FUNCTION_BLOCK "Siemens_vav_compact_controller"   // FB60, SCL
{ S7_Optimized_Access := 'TRUE' }
VERSION : 0.1
   VAR_INPUT
      mb_addr : UInt;
      sp : Real;   // setpoint
      sp_backup : Real;
   END_VAR
   VAR_IN_OUT
      mb_query : "mb_query";
   END_VAR
   VAR
      sb : "mb_station_block_udt";
      read : Struct
         Actual_position : Int;
         Actual_Flow_rel : UInt;
         Actual_Flow_abs : UInt;
         Actual_Pressure : UInt;
      END_STRUCT;
      write1 : Struct
         Setpoint : Int;
      END_STRUCT;
      write2 : Struct
         backup_mode : Int;
         backup_position : Int;
      END_STRUCT;
   END_VAR
BEGIN
   // Siemens - VAV compact controller 
   // GDB181.1E/MO Operating voltage AC 24 V, 5 Nm
   // GLB181.1E/MO Operating voltage AC 24 V, 10 Nm

   // https://www.micromatic.no/globalassets/inriver/resources/
   // bruksanvisning_ko1320-28.pdf

   "mb_station_block_header"(sb := #sb, mb_query := #mb_query);
   #mb_query.mb_addr := #mb_addr;

   #mb_query.mode := #mb_query.c.read.holding_reg;
   #mb_query(data_addr := 3, data_ptr := #read);

   #mb_query.mode := #mb_query.c.write.holding_reg;
   #write1.Setpoint := REAL_TO_INT(#sp) * 100;
   #mb_query(data_addr := 1, data_ptr := #write1);
   #write2.backup_position := REAL_TO_INT(#sp_backup) * 100;
   #mb_query(data_addr := 513, data_ptr := #write2);

   "mb_station_block_footer"(sb := #sb, mb_query := #mb_query);

   (*
   Backup mode (write 2)
   0 = Go to BackupPosition
   1 = Keep last position
   2 = Disabled
   *)
END_FUNCTION_BLOCK

FUNCTION_BLOCK "Siemens_SIWAREX_WP251"   // FB93, SCL
{ S7_Optimized_Access := 'TRUE' }
VERSION : 0.1
   VAR_INPUT
      mb_addr : UInt;
   END_VAR
   VAR_IN_OUT
      mb_query : "mb_query";
   END_VAR
   VAR
      sb : "mb_station_block_udt";
      read1 : Struct
         Unit_of_weight : UInt;   // x1000
         Gross_identifier : UInt;
         Code_for_regulations : UInt;
         Reserve : UInt;
         weighing_range_min : UInt;
         weighing_range_max : Real;
         Calibration_weight : Array[0..2] of Real;
         Calibration_digits : Array[0..2] of Real;
         Scale_interval : Array[0..2] of Real;   // (Page 64)
      END_STRUCT;
      read2 : Struct
         stat : Struct
            x08 : Bool;
            x09 : Bool;
            x10 : Bool;
            x11 : Bool;
            x12 : Bool;
            x13 : Bool;
            x14 : Bool;
            x15 : Bool;
            x00 : Bool;
            x01 : Bool;
            x02 : Bool;
            x03 : Bool;
            x04 : Bool;
            x05 : Bool;
            x06 : Bool;
            x07 : Bool;
         END_STRUCT;
         Reserve : UInt;
         Max_tare_load : Real;
         Max_negative_zero_limit_power_on : Real;
         Max_positive_zero_limit_power_on : Real;
         Max_negative_zero_limit_semi_automatically : Real;
         Max_positive_zero_limit_semi_automatically : Real;
      END_STRUCT;
      read3 : Struct
         standstill : Array[1..2] of Struct
            range : Real;
            "time" : Time;
            max_waiting_time : Time;
         END_STRUCT;
         frequency_low_pass_filter1 : Real;
         Order_no_low_pass_filter1 : UInt;
         depth_average_filter : UInt;
         reserve_1 : UInt;
         weighing_operating_mode : UInt;
         resolution_of_master_totalizer : Real;
         Reserve_2 : Real;
         SecureDisplay_including_weighing_range_data : UInt;
      END_STRUCT;
      read4 : Struct
         SecureDisplay_interface : UInt;   // (Page 71)
         String_header_version_SecureDisplay : String[2];
         SecureDisplay_version : String[12];
         Minimum_zoom_factor_of_SecureDisplay : UInt;
         Reserve_1 : Array[1..3] of Real;
         Reserve_2 : Array[1..3] of UInt;
         Grid_frequency : UInt;   // 0: 50 Hz, 1: 60Hz
      END_STRUCT;
      write1 : Struct
         Smallest_weight_below_TU2 : Real;
         Highest_weight_above_TH2 : Real;
         Single_setpoin : Real;
         Net_weight_average_value : Real;
         Standard_deviation : Real;
      END_STRUCT;
   END_VAR
BEGIN
   // Siemens - SIWAREX WP251 - Electronic Weighing System
   // A5E37203357A
   // 
   // https://cache.industry.siemens.com/dl/files/751/109481751/att_893477/v1/Manual_SIWAREX_WP251_en_en-US.pdf

   "mb_station_block_header"(sb := #sb, mb_query := #mb_query);
   #mb_query.mb_addr := #mb_addr;

   #mb_query.mode := #mb_query.c.read.holding_reg;
   #mb_query(data_addr := 1011, data_ptr := #read1);
   #mb_query(data_addr := 1032, data_ptr := #read2);
   #mb_query(data_addr := 1044, data_ptr := #read3);
   #mb_query(data_addr := 1067, data_ptr := #read4);

   #mb_query.mode := #mb_query.c.write.holding_reg;
   #mb_query(data_addr := 4101, data_ptr := #write1);

   "mb_station_block_footer"(sb := #sb, mb_query := #mb_query);

   (*
   Unit of weight:
   0: "mg"
   1: "g"
   2: "kg"
   3: "t"
   4: "oz" (ounce)
   5: "lb" (pound)
   6: "T" (=short tons)
   7: "TL" (= long tons)

   Gross identifier:
   0: "brutto" 
   1: "Gross"

   Code for regulations:
   0: None
   1: OIML

   Weighing operating mode (Page 71):
   0: NAWI – Filling
   1: NAWI – Removal
   10: AWI
   20: ACI – Filling 
   21: ACI – Removal

   *)
END_FUNCTION_BLOCK

// folder: Library/Modbus/Station blocks/sb untested/Swan

FUNCTION_BLOCK "Swan_AMI_CACE"   // FB65, SCL
{ S7_Optimized_Access := 'TRUE' }
VERSION : 0.1
   VAR_INPUT
      mb_addr : USInt;
   END_VAR
   VAR_IN_OUT
      mb_query : "mb_query";
   END_VAR
   VAR
      sb : "mb_station_block_udt";
      data : Struct
         cond_sc : Array[1..3] of Real;   // µS
         Temp : Array[1..3] of Real;
         flow : Real;
         pH : Real;
         alkalyzer : Real;
         cond_uc : Array[1..3] of Real;
         Pt1000_Temp : Array[1..3] of Real;
         raw_flow : Real;
         case_temperature : Real;
         EDI_voltage : Real;
         EDI_current : Real;
         Degasser_temperature : Real;
         Degasser_boiling_point : Real;
         Degasser_PWM : Real;
         Degasser_line_voltage : Real;
         Degasser_air_pressure : Real;
         Degasser_Case_Temp : Real;
         signal_output : Array[1..2] of Real;
         "Instrument Display Status" : DWord;
      END_STRUCT;
      alarm : Struct
         x00_Cond_1_Alarm_high : Bool;
         x01_Cond_1_Alarm_low : Bool;
         x02_Cond_2_Alarm_high : Bool;
         x03_Cond_2_Alarm_low : Bool;
         x04_Cond_3_Alarm_high : Bool;
         x05_Cond_3_Alarm_low : Bool;
         x06_Temp_1_high : Bool;
         x07_Temp_1_low : Bool;
         x08_sample_flow_high : Bool;
         x09_sample_flow_low : Bool;
         x10_temp_1_shorted : Bool;
         x11_temp_1_disconnected : Bool;
         x12_case_temp_high : Bool;
         x13_case_temp_low : Bool;
         x14_pH_Error : Bool;
         x15_Degasser_frontend : Bool;
         x16_control_timeout : Bool;
         x17_Degasser_disconnected : Bool;
         x18_Temp_2_shorted : Bool;
         x19_Temp_2_disconnected : Bool;
         x20_Temp_3_shorted : Bool;
         x21_Temp_3_disconnected : Bool;
         x22_Degasser_Ctl_Timeout : Bool;
         x23_Input_Active : Bool;
         x24_IC_MK41T56 : Bool;
         x25_IC_LM75 : Bool;
         x26_IC_PCF8574 : Bool;
         x27_Signal_output_open : Bool;
         x28_Calibration_Degasser : Bool;
         x29_EEprom_Front_end : Bool;
         x30_Calibration_Recout : Bool;
         x31_Wrong_Front_end : Bool;
         x32_pH_Alarm_high : Bool;
         x33_pH_Alarm_low : Bool;
         x34_Alkali_Alarm_high : Bool;
         x35_Alkali_Alarm_low : Bool;
         x36_Temp_2_high : Bool;
         x37_Temp_2_low : Bool;
         x38_Temp_3_high : Bool;
         x39_Temp_3_low : Bool;
         x40_Degasser_Line_Voltage : Bool;
         x41_Degasser_Temperature : Bool;
         x42_EDI_out_of_range : Bool;
         x43_No_sample_flow : Bool;
         x44_EDI_DAC_disconnected : Bool;
         "x45_ EDI_ADC_disconnected" : Bool;
         x46 : Bool;
         x47_EDI_module_exhausted : Bool;
      END_STRUCT;
      write : Struct
         x0_relay_contacts_1 : Bool;
         x1_relay_contacts_2 : Bool;
         x2 : Bool;
         x3 : Bool;
         x4 : Bool;
         x5 : Bool;
         x6 : Bool;
         x7 : Bool;
      END_STRUCT;
   END_VAR
BEGIN
   // Swan - AMI CACE - Conductivity measurement 
   // Swan analytical instruments
   // http://www.swan.ch/GetAttachment.axd?attaName=e82f8e94-ab32-4930-8c9d-a56dc0847f61
   // Page 9

   "mb_station_block_header"(sb := #sb,
                             mb_query := #mb_query);
   #mb_query.mb_addr := #mb_addr;
   #mb_query.data_addr := 0;

   #mb_query(mode := #mb_query.c.read.input_reg,
             data_ptr := #data);

   #mb_query(mode := #mb_query.c.read.discrete_input,
             data_ptr := #alarm);

   (*#mb_query(mode := #mb_query.c.write.discrete_output,
             data_len := 2,
             data_ptr := #write);*)

   "mb_station_block_footer"(sb := #sb,
                             mb_query := #mb_query);
END_FUNCTION_BLOCK

FUNCTION_BLOCK "Swan_AMI_Codes-II_CC"   // FB66, SCL
{ S7_Optimized_Access := 'TRUE' }
VERSION : 0.1
   VAR_INPUT
      mb_addr : USInt;
   END_VAR
   VAR_IN_OUT
      mb_query : "mb_query";
   END_VAR
   VAR
      sb : "mb_station_block_udt";
      data : Struct
         free_available_chlorine : Real;   // ppm
         total_chlorine_1_tc1 : Real;   // ppm
         total_chlorine_2_tc2 : Real;   // ppm
         calculated_monochloramine : Real;   // ppm
         calculated_combined_chlorine : Real;   // ppm
         calculated_dichloramine : Real;   // ppm
         temperature : Real;   // °C
         flow : Real;   // B/s
         pH : Real;   // pH
         absorbance : Real;
         photometer_frequency : Real;   // Hz
         remaining_DPD_buffer : Real;   // %
         remaining_potassium_Iodide : Real;   // %
         remaining_cleaning_solution : Real;   // %
         raw_temp_NTK5 : Real;   // Ohm
         raw_flow : Real;   // Hz
         raw_pH : Real;   // mV
         case_temperature : Real;   // °C
         signal_output_1 : Real;   // mA
         signal_output_2 : Real;   // mA
         instrument_display_status : Real;
      END_STRUCT;
      alarm : Struct
         x00_high_fac : Bool;
         x01_low_fac : Bool;
         x02_high_tc1 : Bool;
         x03_low_tc1 : Bool;
         x04_high_tc2 : Bool;
         x05_low_tc2 : Bool;
         x06_sample_temp_high : Bool;
         x07_sample_temp_low : Bool;
         x08_sample_flow_high : Bool;
         x09_sample_flow_low : Bool;
         x10_Temp_shorted : Bool;
         x11_Temp_disconnected : Bool;
         x12_case_temp_high : Bool;
         x13_case_temp_low : Bool;
         x14_valve_1_defective : Bool;
         x15_dis_invalid : Bool;
         x16_control_timeout : Bool;
         x17_reagent_pump : Bool;
         x18_photometer_not_connected : Bool;
         x19_photometer_dirty : Bool;
         x20_absorbance_too_high : Bool;
         x21_reagent_empty : Bool;
         x22_cleaning_reagent : Bool;
         x23_input_active : Bool;
         x24_IC_MK41T56 : Bool;
         x25_IC_LM75 : Bool;
         x26_IC_PCF8574 : Bool;
         x27_signal_output_open : Bool;
         x28_EEprom_motherboard : Bool;
         x29_EEprom_front_end : Bool;
         x30_calibration_recout : Bool;
         x31_wrong_front_end : Bool;
         x32_high_cmc : Bool;
         x33_low_cmc : Bool;
         x34_high_ccc : Bool;
         x35_low_ccc : Bool;
         x36_high_cdc : Bool;
         x37_low_cdc : Bool;
         x38_high_pH : Bool;
         x39_low_pH : Bool;
         x40_DPD_buffer : Bool;
         x41_potassium_Iodide : Bool;
         x42_cleaning_solution : Bool;
         x43 : Bool;
         x44 : Bool;
         x45 : Bool;
         x46 : Bool;
         x47 : Bool;
      END_STRUCT;
      write : Struct
         x0_relay_contacts_1 : Bool;
         x1_relay_contacts_2 : Bool;
         x2_hold : Bool;
         x3_Remote_off : Bool;
         x4 : Bool;
         x5 : Bool;
         x6 : Bool;
         x7 : Bool;
      END_STRUCT;
   END_VAR
BEGIN
   // Swan - AMI Codes-II CC
   //
   // http://www.swan.ch/GetAttachment.axd?attaName=e82f8e94-ab32-4930-8c9d-a56dc0847f61
   // Page 17

   "mb_station_block_header"(sb := #sb,
                             mb_query := #mb_query);
   #mb_query.mb_addr := #mb_addr;
   #mb_query.data_addr := 0;

   #mb_query(mode := #mb_query.c.read.input_reg,
             data_ptr := #data);

   #mb_query(mode := #mb_query.c.read.discrete_input,
             data_ptr := #alarm);

   (*#mb_query(mode := #mb_query.c.write.discrete_output,
             data_len := 4,
             data_ptr := #write);*)

   "mb_station_block_footer"(sb := #sb,
                             mb_query := #mb_query);
END_FUNCTION_BLOCK

FUNCTION_BLOCK "Swan_AMI_Hydrogen"   // FB67, SCL
{ S7_Optimized_Access := 'TRUE' }
VERSION : 0.1
   VAR_INPUT
      mb_addr : USInt;
   END_VAR
   VAR_IN_OUT
      mb_query : "mb_query";
   END_VAR
   VAR
      sb : "mb_station_block_udt";
      data : Struct
         hydrogen : Real;   // ppb
         temperature : Real;   // °C
         flow : Real;   // l/h
         saturation : Real;   // %
         air_pressure : Real;   // hPa
         raw_Current_temp_compensated : Real;   // nA
         raw_current_uncompensated : Real;   // nA
         raw_temp_Pt1000 : Real;   // Ω
         raw_flow : Real;   // Hz
         reserved : Real;
         case_temperature : Real;   // °C
         signal_output_1 : Real;   // mA
         signal_output_2 : Real;   // mA
         instrument_display_status : UDInt;
      END_STRUCT;
      alarm : Struct
         x00_hydrogen_alarm_high : Bool;
         x01_hydrogen_alarm_low : Bool;
         x02_saturation_alarm_high : Bool;
         x03_saturation_alarm_low : Bool;
         x04 : Bool;
         x05 : Bool;
         x06_sample_temp_high : Bool;
         x07_sample_temp_low : Bool;
         x08_sample_flow_high : Bool;
         x09_sample_flow_low : Bool;
         x10_temp_shorted : Bool;
         x11_temp_disconnected : Bool;
         x12_case_temp_high : Bool;
         x13_case_temp_low : Bool;
         x14 : Bool;
         x15 : Bool;
         x16_control_timeout : Bool;
         x17_faraday_efficiency_QED : Bool;
         x18_quality_assurance : Bool;
         x19 : Bool;
         x20 : Bool;
         x21 : Bool;
         x22 : Bool;
         x23_input_active : Bool;
         x24_IC_MK41T56 : Bool;
         x25_IC_LM75 : Bool;
         x26_IC_PCF8574 : Bool;
         x27_Signal_output_open : Bool;
         x28_EEprom_Motherboard : Bool;
         x29_EEprom_Front_end : Bool;
         x30_Calibration_Recout : Bool;
         x31_Wrong_Front_end : Bool;
         x32 : Bool;
         x33 : Bool;
         x34 : Bool;
         x35 : Bool;
         x36 : Bool;
         x37 : Bool;
         x38 : Bool;
         x39 : Bool;
         x40 : Bool;
         x41 : Bool;
         x42 : Bool;
         x43 : Bool;
         x44 : Bool;
         x45 : Bool;
         x46 : Bool;
         x47_Status_Electrolyte_depleted : Bool;
      END_STRUCT;
      write : Struct
         x0_relay_contacts_1 : Bool;
         x1_relay_contacts_2 : Bool;
         x2_hold : Bool;
         x3_Remote_off : Bool;
         x4 : Bool;
         x5 : Bool;
         x6 : Bool;
         x7 : Bool;
      END_STRUCT;
   END_VAR
BEGIN
   // Swan - AMI Hydrogen
   // Swan analytical instruments
   // http://www.swan.ch/GetAttachment.axd?attaName=e82f8e94-ab32-4930-8c9d-a56dc0847f61
   // Page 37

   "mb_station_block_header"(sb := #sb,
                             mb_query := #mb_query);
   #mb_query.mb_addr := #mb_addr;
   #mb_query.data_addr := 0;

   #mb_query(mode := #mb_query.c.read.input_reg,
             data_ptr := #data);

   #mb_query(mode := #mb_query.c.read.discrete_input,
             data_ptr := #alarm);

   (*#mb_query(mode := #mb_query.c.write.discrete_output,
             data_len := 4,
             data_ptr := #write);*)

   "mb_station_block_footer"(sb := #sb,
                             mb_query := #mb_query);
END_FUNCTION_BLOCK

FUNCTION_BLOCK "Swan_AMI_Oxysafe"   // FB68, SCL
{ S7_Optimized_Access := 'TRUE' }
VERSION : 0.1
   VAR_INPUT
      mb_addr : USInt;
   END_VAR
   VAR_IN_OUT
      mb_query : "mb_query";
   END_VAR
   VAR
      sb : "mb_station_block_udt";
      data : Struct
         oxygen : Real;   // ppm
         temperature : Real;   // °C
         flow : Real;   // l/h
         saturation : Real;   // %
         air_pressure : Real;   // hPa
         raw_Oxygen_temp_compensated : Real;   // nA
         raw_oxygen_temp_uncompensated : Real;   // nA
         raw_Temp_Pt1000 : Real;   // Ohm
         raw_flow : Real;   // Hz
         remaining_electrolyte : Real;   // %
         case_temperature : Real;   // °C
         signal_output_1 : Real;   // mA
         signal_output_2 : Real;   // mA
         instrument_display_status : DWord;
      END_STRUCT;
      alarm : Struct
         x00_Oxygen_alarm_high : Bool;
         x01_Oxygen_alarm_low : Bool;
         x02_Saturation_alarm_high : Bool;
         x03_Saturation_alarm_low : Bool;
         x04 : Bool;
         x05 : Bool;
         x06_Sample_temp_high : Bool;
         x07_Sample_temp_low : Bool;
         x08_sample_flow_high : Bool;
         x09_sample_flow_low : Bool;
         x10_temp_shorted : Bool;
         x11_temp_disconnected : Bool;
         x12_case_temp_high : Bool;
         x13_case_temp_low : Bool;
         x14 : Bool;
         x15 : Bool;
         x16_control_timeout : Bool;
         x17_Faraday_efficiency_QED : Bool;
         x18 : Bool;
         x19 : Bool;
         x20 : Bool;
         x21 : Bool;
         x22 : Bool;
         x23_input_active : Bool;
         x24_IC_MK41T56 : Bool;
         x25_IC_LM75 : Bool;
         x26_IC_PCF8574 : Bool;
         x27_Signal_output_open : Bool;
         x28_EEprom_Motherboard : Bool;
         x29_EEprom_Front_end : Bool;
         x30_Calibration_Recout : Bool;
         x31_Wrong_Front_end : Bool;
         x32 : Bool;
         x33 : Bool;
         x34 : Bool;
         x35 : Bool;
         x36 : Bool;
         x37 : Bool;
         x38 : Bool;
         x39 : Bool;
         x40_Electrolyte_depleted : Bool;
         x41 : Bool;
         x42 : Bool;
         x43 : Bool;
         x44 : Bool;
         x45 : Bool;
         x46 : Bool;
         x47 : Bool;
      END_STRUCT;
      write : Struct
         x0_relay_contacts_1 : Bool;
         x1_relay_contacts_2 : Bool;
         x2_hold : Bool;
         x3_Remote_off : Bool;
         x4 : Bool;
         x5 : Bool;
         x6 : Bool;
         x7 : Bool;
      END_STRUCT;
   END_VAR
BEGIN
   // Swan - AMI - Oxysafe
   // Swan analytical instruments
   // http://www.swan.ch/GetAttachment.axd?attaName=e82f8e94-ab32-4930-8c9d-a56dc0847f61
   // Page 53

   "mb_station_block_header"(sb := #sb,
                             mb_query := #mb_query);
   #mb_query.mb_addr := #mb_addr;
   #mb_query.data_addr := 0;

   #mb_query(mode := #mb_query.c.read.input_reg,
             data_ptr := #data);

   #mb_query(mode := #mb_query.c.read.discrete_input,
             data_ptr := #alarm);

   (*#mb_query(mode := #mb_query.c.write.discrete_output,
             data_len := 4,
             data_ptr := #write);*) 

   "mb_station_block_footer"(sb := #sb,
                             mb_query := #mb_query);
END_FUNCTION_BLOCK

FUNCTION_BLOCK "Swan_AMI_pH-Redox"   // FB69, SCL
{ S7_Optimized_Access := 'TRUE' }
VERSION : 0.1
   VAR_INPUT
      mb_addr : USInt;
   END_VAR
   VAR_IN_OUT
      mb_query : "mb_query";
   END_VAR
   VAR
      sb : "mb_station_block_udt";
      data : Struct
         pH_Redox : Real;   // pH/mV
         temperature : Real;   // °C
         Flow : Real;   // l/h
         raw_signal : Real;   // mV
         Pt_1000_temp : Real;   // ohm
         raw_flow : Real;   // Hz
         sensor_check : Real;   // Mohm
         case_temperature : Real;   // °C
         signal_output_1 : Real;   // mA
         signal_output_2 : Real;   // mA
         instrument_display_status : DWord;
      END_STRUCT;
      alarm : Struct
         x00_alarm_high : Bool;
         x01_alarm_low : Bool;
         x02 : Bool;
         x03 : Bool;
         x04 : Bool;
         x05 : Bool;
         x06_sample_temp_high : Bool;
         x07_sample_temp_low : Bool;
         x08_sample_flow_high : Bool;
         x09_sample_flow_low : Bool;
         x10_temp_shorted : Bool;
         x11_temp_disconnected : Bool;
         x12_case_temp_high : Bool;
         x13_case_temp_low : Bool;
         x14 : Bool;
         x15 : Bool;
         x16_control_timeout : Bool;
         x17 : Bool;
         x18 : Bool;
         x19 : Bool;
         x20 : Bool;
         x21 : Bool;
         x22 : Bool;
         x23_input_active : Bool;
         x24_IC_MK41T56 : Bool;
         x25_IC_LM75 : Bool;
         x26_IC_PCF8574 : Bool;
         x27_Signal_output_open : Bool;
         x28_EEprom_Motherboard : Bool;
         x29_EEprom_Front_end : Bool;
         x30_Calibration_Recout : Bool;
         x31_Wrong_Front_end : Bool;
      END_STRUCT;
      write : Struct
         x0_relay_contacts_1 : Bool;
         x1_relay_contacts_2 : Bool;
         x2_hold : Bool;
         x3_Remote_off : Bool;
         x4 : Bool;
         x5 : Bool;
         x6 : Bool;
         x7 : Bool;
      END_STRUCT;
   END_VAR
BEGIN
   // Swan - AMI pH-Redox
   // Swan analytical instruments
   // 
   // http://www.swan.ch/GetAttachment.axd?attaName=e82f8e94-ab32-4930-8c9d-a56dc0847f61
   // Page 73

   "mb_station_block_header"(sb := #sb, mb_query := #mb_query);
   #mb_query.mb_addr := #mb_addr;
   #mb_query.data_addr := 0;

   #mb_query(mode := #mb_query.c.read.input_reg,
             data_ptr := #data);

   #mb_query(mode := #mb_query.c.read.discrete_input,
             data_ptr := #alarm);

   (*#mb_query(mode := #mb_query.c.write.discrete_output,
             data_len := 4,
             data_ptr := #write);*)

   "mb_station_block_footer"(sb := #sb, mb_query := #mb_query);
END_FUNCTION_BLOCK

// folder: Library/Modbus/Station blocks/z Extend blocks

FUNCTION_BLOCK "searchDevice"   // FB41, SCL
{ S7_Optimized_Access := 'TRUE' }
VERSION : 0.1
   VAR_OUTPUT
      Done : Bool;
      No_finding : Bool;
   END_VAR
   VAR_IN_OUT
      start_search : Bool;
      mb_addr : UInt;
      mb_query : "mb_query";
   END_VAR
   VAR
      reset_at_start : Bool;
      data_addr : UDInt;
      _ : Bool;
      rtirg_start : R_TRIG;
      resualt_data : Word;
   END_VAR
BEGIN
   #rtirg_start(CLK := #start_search);
   IF #rtirg_start.Q AND #reset_at_start THEN
       #mb_addr := 1;
   END_IF;

   IF #start_search THEN
       #Done := false;
       #No_finding := false;
       #mb_query(mb_addr := #mb_addr,
                 mode := #mb_query.c.read.holding_reg,
                 data_addr := #data_addr,
                 data_ptr := #resualt_data);
       IF #mb_query.Done
           OR #mb_query.Error AND NOT #mb_query.stat.error_comm
       THEN
           #Done := true;
           #start_search := false;
       ELSIF #mb_query.Error THEN
           IF #mb_addr < 247 THEN
               #mb_addr += 1;
           ELSE
               #No_finding := true;
               #start_search := false;
           END_IF;
       END_IF;
   END_IF;
END_FUNCTION_BLOCK